FUNCTION_BLOCK "ST10_Flow14_B2Press"
VAR_INPUT
  iSysInface : "RCS_SysComInterface_V1";
END_VAR
VAR_IN_OUT
  ioPM_Inface : "RCS_PMInterface_V1";
  ioStatus : Int;
END_VAR
VAR
  sCtrlMode : "SysFlowCtrlGraph";
  sUpdMES_Data : Bool;
  "工件放行中" : Bool;
  "前站站号" : UInt;
  "本站站号" : UInt;
  "弹窗Temp" : Array[1..10] of Int;
  AlarmID : Int;
  TON : Array[0..10] of TON_TIME;
  TOF : Array[0..10] of TOF_TIME;
  sUP : Array[0..10] of Bool;
  "更新RFID完成" : Bool;
  RT_DATA : G7_RTDataPlus_V6;
  Trans1 : G7_TransitionPlus_V6;
  Trans2 : G7_TransitionPlus_V6;
  Trans3 : G7_TransitionPlus_V6;
  Trans325 : G7_TransitionPlus_V6;
  Trans10 : G7_TransitionPlus_V6;
  Trans7 : G7_TransitionPlus_V6;
  Trans102 : G7_TransitionPlus_V6;
  Trans12 : G7_TransitionPlus_V6;
  Trans15 : G7_TransitionPlus_V6;
  Trans17 : G7_TransitionPlus_V6;
  Trans18 : G7_TransitionPlus_V6;
  Trans19 : G7_TransitionPlus_V6;
  Trans20 : G7_TransitionPlus_V6;
  Trans21 : G7_TransitionPlus_V6;
  Trans22 : G7_TransitionPlus_V6;
  Trans23 : G7_TransitionPlus_V6;
  Trans24 : G7_TransitionPlus_V6;
  Trans25 : G7_TransitionPlus_V6;
  Trans28 : G7_TransitionPlus_V6;
  Trans29 : G7_TransitionPlus_V6;
  Trans30 : G7_TransitionPlus_V6;
  Trans9 : G7_TransitionPlus_V6;
  Trans31 : G7_TransitionPlus_V6;
  Trans32 : G7_TransitionPlus_V6;
  Trans33 : G7_TransitionPlus_V6;
  Trans34 : G7_TransitionPlus_V6;
  Trans35 : G7_TransitionPlus_V6;
  Trans36 : G7_TransitionPlus_V6;
  Trans200 : G7_TransitionPlus_V6;
  Empty : G7_TransitionPlus_V6;
  Trans266 : G7_TransitionPlus_V6;
  Trans11 : G7_TransitionPlus_V6;
  Trans249 : G7_TransitionPlus_V6;
  Trans283 : G7_TransitionPlus_V6;
  Trans284 : G7_TransitionPlus_V6;
  Trans199 : G7_TransitionPlus_V6;
  Trans765 : G7_TransitionPlus_V6;
  Trans117 : G7_TransitionPlus_V6;
  Trans766 : G7_TransitionPlus_V6;
  Trans119 : G7_TransitionPlus_V6;
  Trans120 : G7_TransitionPlus_V6;
  Trans767 : G7_TransitionPlus_V6;
  Trans236 : G7_TransitionPlus_V6;
  Trans124 : G7_TransitionPlus_V6;
  Trans125 : G7_TransitionPlus_V6;
  Trans128 : G7_TransitionPlus_V6;
  Trans129 : G7_TransitionPlus_V6;
  Trans130 : G7_TransitionPlus_V6;
  Trans768 : G7_TransitionPlus_V6;
  Trans132 : G7_TransitionPlus_V6;
  Trans133 : G7_TransitionPlus_V6;
  Trans134 : G7_TransitionPlus_V6;
  Trans135 : G7_TransitionPlus_V6;
  Trans136 : G7_TransitionPlus_V6;
  Trans138 : G7_TransitionPlus_V6;
  Trans140 : G7_TransitionPlus_V6;
  HavePart : G7_TransitionPlus_V6;
  Trans303 : G7_TransitionPlus_V6;
  Trans304 : G7_TransitionPlus_V6;
  Trans142 : G7_TransitionPlus_V6;
  Trans137 : G7_TransitionPlus_V6;
  Trans144 : G7_TransitionPlus_V6;
  Trans145 : G7_TransitionPlus_V6;
  Trans146 : G7_TransitionPlus_V6;
  Trans148 : G7_TransitionPlus_V6;
  Trans139 : G7_TransitionPlus_V6;
  Trans147 : G7_TransitionPlus_V6;
  Trans201 : G7_TransitionPlus_V6;
  Trans211 : G7_TransitionPlus_V6;
  Trans250 : G7_TransitionPlus_V6;
  Trans252 : G7_TransitionPlus_V6;
  Trans262 : G7_TransitionPlus_V6;
  Trans257 : G7_TransitionPlus_V6;
  Trans258 : G7_TransitionPlus_V6;
  Trans261 : G7_TransitionPlus_V6;
  Trans263 : G7_TransitionPlus_V6;
  Trans265 : G7_TransitionPlus_V6;
  Trans267 : G7_TransitionPlus_V6;
  Trans269 : G7_TransitionPlus_V6;
  Trans259 : G7_TransitionPlus_V6;
  Trans302 : G7_TransitionPlus_V6;
  Trans26 : G7_TransitionPlus_V6;
  Trans16 : G7_TransitionPlus_V6;
  Trans316 : G7_TransitionPlus_V6;
  Trans311 : G7_TransitionPlus_V6;
  Trans312 : G7_TransitionPlus_V6;
  Trans313 : G7_TransitionPlus_V6;
  Online : G7_TransitionPlus_V6;
  Trans317 : G7_TransitionPlus_V6;
  Trans318 : G7_TransitionPlus_V6;
  Trans319 : G7_TransitionPlus_V6;
  Trans315 : G7_TransitionPlus_V6;
  Trans320 : G7_TransitionPlus_V6;
  Trans322 : G7_TransitionPlus_V6;
  Online_1 : G7_TransitionPlus_V6;
  Trans260 : G7_TransitionPlus_V6;
  Trans323 : G7_TransitionPlus_V6;
  Trans324 : G7_TransitionPlus_V6;
  Trans326 : G7_TransitionPlus_V6;
  Trans327 : G7_TransitionPlus_V6;
  Trans328 : G7_TransitionPlus_V6;
  Trans321 : G7_TransitionPlus_V6;
  Trans224 : G7_TransitionPlus_V6;
  OK : G7_TransitionPlus_V6;
  Trans403 : G7_TransitionPlus_V6;
  Trans405 : G7_TransitionPlus_V6;
  NG : G7_TransitionPlus_V6;
  Trans404 : G7_TransitionPlus_V6;
  Trans412 : G7_TransitionPlus_V6;
  Trans407 : G7_TransitionPlus_V6;
  Trans619 : G7_TransitionPlus_V6;
  Trans600 : G7_TransitionPlus_V6;
  Trans290 : G7_TransitionPlus_V6;
  Trans699 : G7_TransitionPlus_V6;
  Trans613 : G7_TransitionPlus_V6;
  Alarm : G7_TransitionPlus_V6;
  F14_Initial : G7_StepPlus_V6;
  S2 : G7_StepPlus_V6;
  S3 : G7_StepPlus_V6;
  S4 : G7_StepPlus_V6;
  S5_MESInitial : G7_StepPlus_V6;
  PressProgram : G7_StepPlus_V6;
  PressHoming : G7_StepPlus_V6;
  S10_InitialFinish : G7_StepPlus_V6;
  "PressReady?" : G7_StepPlus_V6;
  "PressHoming?" : G7_StepPlus_V6;
  Step14 : G7_StepPlus_V6;
  CheckPressGripStatus : G7_StepPlus_V6;
  ShaftAndRingOK : G7_StepPlus_V6;
  "Press NG" : G7_StepPlus_V6;
  MES : G7_StepPlus_V6;
  MESOK : G7_StepPlus_V6;
  PressProgram_1 : G7_StepPlus_V6;
  PressHoming_1 : G7_StepPlus_V6;
  "PressReady?_1" : G7_StepPlus_V6;
  "PressHoming?_1" : G7_StepPlus_V6;
  Step15 : G7_StepPlus_V6;
  MES_1NG : G7_StepPlus_V6;
  ProcessStart : G7_StepPlus_V6;
  "Determine product status" : G7_StepPlus_V6;
  CheckMachineStatus : G7_StepPlus_V6;
  "Normal mode" : G7_StepPlus_V6;
  "ProcessStart,CTStart" : G7_StepPlus_V6;
  "Request robot putShaft" : G7_StepPlus_V6;
  "Request robot putRing" : G7_StepPlus_V6;
  "RobotLeavePress Area" : G7_StepPlus_V6;
  "B-PressFitting-01GripperCylinderToHP" : G7_StepPlus_V6;
  CheckRingExist : G7_StepPlus_V6;
  "Status Alarm" : G7_StepPlus_V6;
  "B-PressFitting-01GripperCylinderToWP" : G7_StepPlus_V6;
  "B-PressFitting-01CylinderToHP" : G7_StepPlus_V6;
  RobotLeavePressArea : G7_StepPlus_V6;
  PartStatus : G7_StepPlus_V6;
  ShaftOK : G7_StepPlus_V6;
  StatusAlarm : G7_StepPlus_V6;
  PutRing : G7_StepPlus_V6;
  NoPart : G7_StepPlus_V6;
  "Wait  robot finish task" : G7_StepPlus_V6;
  "Wait robot finish task" : G7_StepPlus_V6;
  DataMove : G7_StepPlus_V6;
  "Wait robot in safety area" : G7_StepPlus_V6;
  "Wait  robot finish task_1" : G7_StepPlus_V6;
  PartStatus_1 : G7_StepPlus_V6;
  CheckPressSensor : G7_StepPlus_V6;
  CheckPressProgram : G7_StepPlus_V6;
  "B-PressFitting-01CylinderToHP_1" : G7_StepPlus_V6;
  StartCycle : G7_StepPlus_V6;
  ResetPressStart : G7_StepPlus_V6;
  "ProcessFInish 1" : G7_StepPlus_V6;
  CheckPressResult : G7_StepPlus_V6;
  ResultOKData : G7_StepPlus_V6;
  ResultNGData : G7_StepPlus_V6;
  Step147 : G7_StepPlus_V6;
  "MES  Check   In" : G7_StepPlus_V6;
  Pressing : G7_StepPlus_V6;
  WaitPressFinish : G7_StepPlus_V6;
  CheckPressReady : G7_StepPlus_V6;
  "Process FInish" : G7_StepPlus_V6;
  PartCheck : G7_StepPlus_V6;
  "Part Check" : G7_StepPlus_V6;
  ProductCheckAlarm : G7_StepPlus_V6;
  ProductCheckAlarm_1 : G7_StepPlus_V6;
  ResetMesCheckRequest : G7_StepPlus_V6;
  ResetMesUnloadRequest_1 : G7_StepPlus_V6;
  "Prepare MES CheckData" : G7_StepPlus_V6;
  "Prepare MES CheckData_1" : G7_StepPlus_V6;
  MesCheckResult_1 : G7_StepPlus_V6;
  MESOverTime_1 : G7_StepPlus_V6;
  "MES Check NG_2" : G7_StepPlus_V6;
  MesCheckIn_1 : G7_StepPlus_V6;
  CheckFinish_1 : G7_StepPlus_V6;
  Bypass : G7_StepPlus_V6;
  Step313 : G7_StepPlus_V6;
  "MES Check NG_3" : G7_StepPlus_V6;
  Bypass_1 : G7_StepPlus_V6;
  Step314 : G7_StepPlus_V6;
  MESOverTime : G7_StepPlus_V6;
  ok_1 : G7_StepPlus_V6;
  Step400 : G7_StepPlus_V6;
  JudgeStatus : G7_StepPlus_V6;
  OKCount : G7_StepPlus_V6;
  ProcessFinish : G7_StepPlus_V6;
  NGCount : G7_StepPlus_V6;
  "MES Result OK_1" : G7_StepPlus_V6;
  "Request robot pick" : G7_StepPlus_V6;
  "MES Result" : G7_StepPlus_V6;
  "MES Check Finish" : G7_StepPlus_V6;
  RobotPick : G7_StepPlus_V6;
  DataClear : G7_StepPlus_V6;
  ProcessFinsh : G7_StepPlus_V6;
END_VAR
VAR_TEMP
  Tempresult : USInt;
  "本站站号乘10" : UInt;
END_VAR
BEGIN
  // Původní jazyk: GRAPH
  // Zdroj XML: EXPORT/Program blocks/OP010/03_Auto/B_Press/ST10_Flow14_B2Press.xml
  // (Nebylo nalezeno StructuredText/FlgNet/StatementList; logika může být v GRAPH nebo v nepodporované reprezentaci.)
END_FUNCTION_BLOCK
